// TIA Portal V19 export
FUNCTION "PPrf_CALL" : Void   // FC81, LAD
TITLE = PROFILE PROGRAM MANAGEMENT
// stored: SetENOAutomatically false
   VAR_TEMP
      i : Int;
   END_VAR
BEGIN

REGION Network 1: Profile program manager
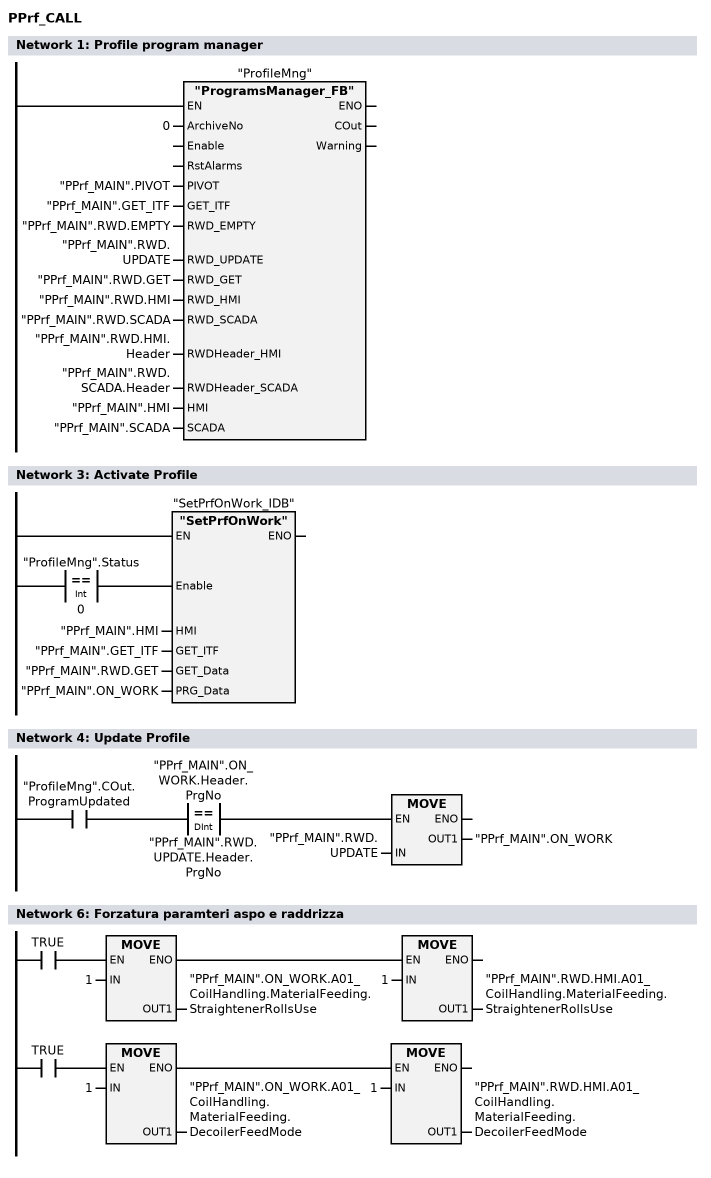
   RUNG wire#powerrail
      "ProfileMng"(ArchiveNo := 0, Enable :=, RstAlarms :=, PIVOT := "PPrf_MAIN".PIVOT, GET_ITF := "PPrf_MAIN".GET_ITF, RWD_EMPTY := "PPrf_MAIN".RWD.EMPTY, RWD_UPDATE := "PPrf_MAIN".RWD.UPDATE, RWD_GET := "PPrf_MAIN".RWD.GET, RWD_HMI := "PPrf_MAIN".RWD.HMI, RWD_SCADA := "PPrf_MAIN".RWD.SCADA, RWDHeader_HMI := "PPrf_MAIN".RWD.HMI.Header, RWDHeader_SCADA := "PPrf_MAIN".RWD.SCADA.Header, HMI := "PPrf_MAIN".HMI, SCADA := "PPrf_MAIN".SCADA, COut =>, Warning =>)
   END_RUNG
   // the same network as SCL:
   "ProfileMng"(ArchiveNo := 0,   // "ProgramsManager_FB"
                PIVOT := "PPrf_MAIN".PIVOT,
                GET_ITF := "PPrf_MAIN".GET_ITF,
                RWD_EMPTY := "PPrf_MAIN".RWD.EMPTY,
                RWD_UPDATE := "PPrf_MAIN".RWD.UPDATE,
                RWD_GET := "PPrf_MAIN".RWD.GET,
                RWD_HMI := "PPrf_MAIN".RWD.HMI,
                RWD_SCADA := "PPrf_MAIN".RWD.SCADA,
                RWDHeader_HMI := "PPrf_MAIN".RWD.HMI.Header,
                RWDHeader_SCADA := "PPrf_MAIN".RWD.SCADA.Header,
                HMI := "PPrf_MAIN".HMI,
                SCADA := "PPrf_MAIN".SCADA);
END_REGION

REGION Network 3: Activate Profile
   RUNG wire#powerrail
      "SetPrfOnWork_IDB"(Enable := wire#w1, HMI := "PPrf_MAIN".HMI, GET_ITF := "PPrf_MAIN".GET_ITF, GET_Data := "PPrf_MAIN".RWD.GET, PRG_Data := "PPrf_MAIN".ON_WORK)
   END_RUNG
   RUNG wire#powerrail
      { S7_Templates := "SrcType := Int" } EQ_Contact(in1 := "ProfileMng".Status, in2 := 0)
   END_RUNG wire#w1
   // the same network as SCL:
   "SetPrfOnWork_IDB"(Enable := "ProfileMng".Status = 0,   // "SetPrfOnWork"
                      HMI := "PPrf_MAIN".HMI,
                      GET_ITF := "PPrf_MAIN".GET_ITF,
                      GET_Data := "PPrf_MAIN".RWD.GET,
                      PRG_Data := "PPrf_MAIN".ON_WORK);
END_REGION

REGION Network 4: Update Profile
   RUNG wire#powerrail
      Contact( "ProfileMng".COut.ProgramUpdated )
      { S7_Templates := "SrcType := DInt" } EQ_Contact(in1 := "PPrf_MAIN".ON_WORK.Header.PrgNo, in2 := "PPrf_MAIN".RWD.UPDATE.Header.PrgNo)
      Move(in := "PPrf_MAIN".RWD.UPDATE, out1 => "PPrf_MAIN".ON_WORK)
   END_RUNG
   // the same network as SCL:
   IF "ProfileMng".COut.ProgramUpdated AND ("PPrf_MAIN".ON_WORK.Header.PrgNo = "PPrf_MAIN".RWD.UPDATE.Header.PrgNo) THEN
       "PPrf_MAIN".ON_WORK := "PPrf_MAIN".RWD.UPDATE;
   END_IF;
END_REGION

REGION Network 5 (SCL): Conversione codice spessore in mm
   "PPrf_MAIN".ON_WORK.GeneralData.Material_Thickness := INT_TO_REAL("PPrf_MAIN".ON_WORK.GeneralData.Beam_TK_Code) / 100.0;
END_REGION

REGION Network 6: Forzatura paramteri aspo e raddrizza
   RUNG wire#powerrail
      Contact( TRUE )
      Move(in := 1, out1 => "PPrf_MAIN".ON_WORK.A01_CoilHandling.MaterialFeeding.StraightenerRollsUse)
      Move(in := 1, out1 => "PPrf_MAIN".RWD.HMI.A01_CoilHandling.MaterialFeeding.StraightenerRollsUse)
   END_RUNG
   RUNG wire#powerrail
      Contact( TRUE )
      Move(in := 1, out1 => "PPrf_MAIN".ON_WORK.A01_CoilHandling.MaterialFeeding.DecoilerFeedMode)
      Move(in := 1, out1 => "PPrf_MAIN".RWD.HMI.A01_CoilHandling.MaterialFeeding.DecoilerFeedMode)
   END_RUNG
   // the same network as SCL:
   IF TRUE THEN
       "PPrf_MAIN".ON_WORK.A01_CoilHandling.MaterialFeeding.StraightenerRollsUse := 1;
       "PPrf_MAIN".RWD.HMI.A01_CoilHandling.MaterialFeeding.StraightenerRollsUse := 1;
       "PPrf_MAIN".ON_WORK.A01_CoilHandling.MaterialFeeding.DecoilerFeedMode := 1;
       "PPrf_MAIN".RWD.HMI.A01_CoilHandling.MaterialFeeding.DecoilerFeedMode := 1;
   END_IF;
END_REGION
END_FUNCTION
